# EPICS autosave request: iocBoot/obsolete/ioc13ide/auto_positions.req
file "CARS_40_motor_positions.req", P=$(P)
